Staubli VAL3: _resetAllPallet.dtx

string sPalletName
mdesc nom_speed = {rmax=9999, blend=off}
